// TIA Portal V18 export
DATA_BLOCK "Function Pressure release"   // DB277
{ S7_Optimized_Access := 'TRUE' }
VERSION : 0.1
// stored: AutoNumber true, DBAccessibleFromOPCUA true, IsOnlyStoredInLoadMemory false, IsRetainMemResEnabled false, IsWriteProtectedInAS false, MemoryReserve 100
   VAR
      "A" : Struct
         Control : Struct
            "Pressure releasing" : Bool;
            "Start release" : Bool;
         END_STRUCT;
         output : Struct
            "ON_outlet Valve A" : Bool;
         END_STRUCT;
      END_STRUCT;
      "B" : Struct
         Control : Struct
            "Start release" : Bool;
            "Pressure releasing" : Bool;
         END_STRUCT;
         output : Struct
            "ON_outlet Valve B" : Bool;
         END_STRUCT;
      END_STRUCT;
      AB : Struct
         Control : Struct
            "Start release" : Bool;
            "Pressure releasing" : Bool;
         END_STRUCT;
         output : Struct
            "ON_outlet Valve B" : Bool;
            "ON_outlet Valve A" : Bool;
         END_STRUCT;
      END_STRUCT;
   END_VAR
BEGIN
END_DATA_BLOCK
